FUNCTION_BLOCK MyCalculatorTests EXTENDS FB_TestSuite
VAR_INPUT
END_VAR
VAR_OUTPUT
END_VAR
VAR
END_VAR

METHOD DivideByZeroTest : REFERENCE TO FB_Test
VAR
	myCalc : MyCalculatorClass;
    Result : UINT;
    ExpectedSum : UINT := 4;
END_VAR
TEST('GivenAZeroDivisorThenTheCalcShouldReturnAError');
 
Result :=  myCalc.Divide(2,0);

AssertEquals(Expected := ExpectedSum,
             Actual := Result,
             Message := 'The division didnt return an error');
 
TEST_FINISHED();
END_METHOD

METHOD TwoPositiveIntegers : REFERENCE TO FB_Test
VAR
	myCalc : MyCalculatorClass;
    Result : INT;
    ExpectedSum : INT := 2;
END_VAR
TEST('GivenTwoPositiveIntegersThenTheResultShouldBeValid');
 
Result := myCalc.Divide(4,2);
 
AssertEquals(Expected := ExpectedSum,
             Actual := Result,
             Message := 'The division returned an error');
 
TEST_FINISHED();
END_METHOD

END_FUNCTION_BLOCK

(* stored: Version 1.1.0.1, ProductVersion 3.1.4024.12
   POU MyCalculatorTests: Id {e1a3d36a-7d44-45ec-aa78-a22fd6fcc456}, SpecialFunc None
   Method DivideByZeroTest: Id {56b81339-bf83-457b-9939-89624932ecb3}
   Method TwoPositiveIntegers: Id {369e8880-8c75-4617-a40e-88d243312c48} *)
